// TIA Portal project "PAD_Printer" (V16)

(* hardware
DEVICE "S7-1200 station_1"  S7-1200 Station
   slot 0: "Rack_0"  S7-1200 Rack  Rack  V1.0
   slot 1: "PLC_1"  CPU 1214C DC/DC/DC  6ES7 214-1AG40-0XB0  V4.4
DEVICE "HMI_1"  TP700 Comfort
   slot 0: "HMI_1"  TP700 Comfort  6AV2 124-0GC01-0AX0  16.0.0.0
   slot 1: "HMI_RT_1"  TP700 Comfort  6AV2 124-0GC01-0AX0  16.0.0.0
   slot 5: "HMI_1.IE_CP_1"  PROFINET Interface  16.0.0.0
      slot 1: "PROFINET Interface_1"  PROFINET Interface
         slot 1: "Port_1"  Port
         slot 2: "Port_2"  Port
   slot 7: "HMI_1.MPI/DP_CP_1"  MPI/DP Interface  16.0.0.0
*)

// ===== PLC "PLC_1"  CPU 1214C DC/DC/DC =====

VAR_GLOBAL   // PLC tag table "Default tag table"
   "AUTO" AT %I0.0 : Bool;   // Chế độ Auto
   "MAN" AT %I0.1 : Bool;   // Chế độ Manual
   "FOOT SWITCH" AT %I0.2 : Bool;   // Bàn đạp của chế độ Manual
   "X-CYLINDER IN" AT %I0.3 : Bool;   // Cảm biến xylanh thu về
   "X-CYLINDER OUT" AT %I0.4 : Bool;   // Cảm biến xylanh đi ra
   "Y-CYLINDER UPPER" AT %I0.5 : Bool;   // Cảm biến xylanh bên trên
   "Y-CYLINDER LOWER" AT %I0.6 : Bool;   // Cảm biến xylanh bên dưới
   "CLEAN" AT %I0.7 : Bool;   // Chế độ Clean
   "X-CYLINDER RUN" AT %Q0.0 : Bool;   // Xylanh trục X chạy
   "Y-CYLINDER RUN" AT %Q0.1 : Bool;   // Xylanh trục Y chạy
   "Tag_1" AT %M5.0 : Bool;   // Bit trung gian của chế độ Manual, Auto
   "Tag_2" AT %M5.1 : Bool;   // Bit trung gian của chế độ Manual, Auto
   "Time_delay" AT %M5.2 : Bool;   // Bit trung gian timer của chế độ Auto
   "Tag_3" AT %M5.3 : Bool;   // Bit trung gian của chế độ Manual
   "Tag_4" AT %M5.4 : Bool;   // Bit trung gian của chế độ Auto
   "Tag_5" AT %M5.5 : Bool;   // Bit trung gian của chế độ Auto
   "Tag_6" AT %M5.6 : Bool;   // Bit trung gian của chế độ Auto
   "PV-T" AT %MD100 : DInt;   // Hiển thị thời gian delay trong Auto
   "Tag_7" AT %M6.0 : Bool;   // Bit nhớ của lệnh xung sườn xuống
   "Tag_8" AT %M6.1 : Bool;   // Bit nhớ của lệnh xung sườn xuống
END_VAR

DATA_BLOCK "DATA"   // DB1
{ S7_Optimized_Access := 'FALSE' }
VERSION : 0.1
   VAR
      AUTO : Bool;   // Chế độ Auto
      MAN : Bool;   // Chế độ Manual
      "FOOT SWITCH" : Bool;   // Bàn đạp của chế độ Manual
      "X-CYLINDER IN" : Bool;   // Cảm biến xylanh thu về
      "X-CYLINDER OUT" : Bool;   // Cảm biến xylanh đi ra
      "Y-CYLINDER UPPER" : Bool;   // Cảm biến xylanh bên trên
      "Y-CYLINDER LOWER" : Bool;   // Cảm biến xylanh bên dưới
      CLEAN : Bool;   // Chế độ Clean
      "X-CYLINDER RUN" : Bool;   // Xylanh trục X chạy
      "Y-CYLINDER RUN" : Bool;   // Xylanh trục Y chạy
      Define_Man : Bool;
      Define_Auto : Bool;
      AUTO_I : Bool;
      MAN_I : Bool;
      "FOOT SWITCH_I" : Bool;
      "X-CYLINDER IN_I" : Bool;
      "X_CYLINDER OUT_I" : Bool;
      "Y-CYLINDER UPPER_I" : Bool;
      "Y-CYLINDER LOWER_I" : Bool;
      CLEAN_I : Bool;
      "X-CYLINDER RUN_I" : Bool;
      "Y-CYLINDER RUN_I" : Bool;
      RESETALL : Bool;
   END_VAR
BEGIN
END_DATA_BLOCK

// folder: System blocks/Program resources

DATA_BLOCK "T"   // DB2
{ S7_Optimized_Access := 'TRUE' }
AUTHOR : Simatic
FAMILY : IEC
NAME : IEC_TMR
VERSION : 1.0
// stored: InstanceOfName IEC_TIMER
"IEC_TIMER"
BEGIN
END_DATA_BLOCK

// folder: (top level)

FUNCTION "INPUT" : Void   // FC1, LAD
{ S7_Optimized_Access := 'TRUE' }
VERSION : 0.1
BEGIN

REGION Network 1: Chế độ AUTO
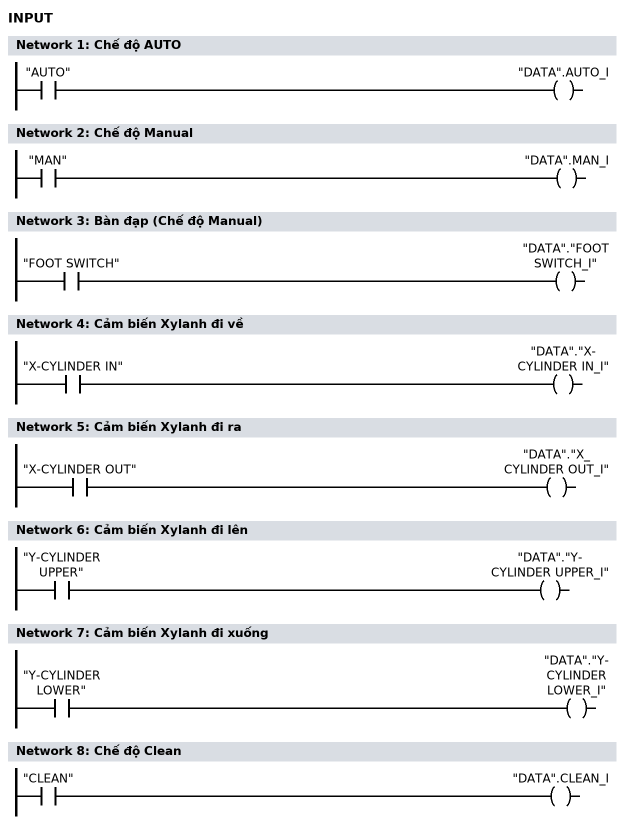
   RUNG wire#powerrail
      Contact( "AUTO" )
      Coil( "DATA".AUTO_I )
   END_RUNG
   // the same network as SCL:
   "DATA".AUTO_I := "AUTO";
END_REGION

REGION Network 2: Chế độ Manual
   RUNG wire#powerrail
      Contact( "MAN" )
      Coil( "DATA".MAN_I )
   END_RUNG
   // the same network as SCL:
   "DATA".MAN_I := "MAN";
END_REGION

REGION Network 3: Bàn đạp (Chế độ Manual)
   RUNG wire#powerrail
      Contact( "FOOT SWITCH" )
      Coil( "DATA"."FOOT SWITCH_I" )
   END_RUNG
   // the same network as SCL:
   "DATA"."FOOT SWITCH_I" := "FOOT SWITCH";
END_REGION

REGION Network 4: Cảm biến Xylanh đi về
   RUNG wire#powerrail
      Contact( "X-CYLINDER IN" )
      Coil( "DATA"."X-CYLINDER IN_I" )
   END_RUNG
   // the same network as SCL:
   "DATA"."X-CYLINDER IN_I" := "X-CYLINDER IN";
END_REGION

REGION Network 5: Cảm biến Xylanh đi ra
   RUNG wire#powerrail
      Contact( "X-CYLINDER OUT" )
      Coil( "DATA"."X_CYLINDER OUT_I" )
   END_RUNG
   // the same network as SCL:
   "DATA"."X_CYLINDER OUT_I" := "X-CYLINDER OUT";
END_REGION

REGION Network 6: Cảm biến Xylanh đi lên
   RUNG wire#powerrail
      Contact( "Y-CYLINDER UPPER" )
      Coil( "DATA"."Y-CYLINDER UPPER_I" )
   END_RUNG
   // the same network as SCL:
   "DATA"."Y-CYLINDER UPPER_I" := "Y-CYLINDER UPPER";
END_REGION

REGION Network 7: Cảm biến Xylanh đi xuống
   RUNG wire#powerrail
      Contact( "Y-CYLINDER LOWER" )
      Coil( "DATA"."Y-CYLINDER LOWER_I" )
   END_RUNG
   // the same network as SCL:
   "DATA"."Y-CYLINDER LOWER_I" := "Y-CYLINDER LOWER";
END_REGION

REGION Network 8: Chế độ Clean
   RUNG wire#powerrail
      Contact( "CLEAN" )
      Coil( "DATA".CLEAN_I )
   END_RUNG
   // the same network as SCL:
   "DATA".CLEAN_I := "CLEAN";
END_REGION
END_FUNCTION

FUNCTION "OUTPUT" : Void   // FC2, LAD
{ S7_Optimized_Access := 'TRUE' }
VERSION : 0.1
BEGIN

REGION Network 1: Chạy Xylanh trục X
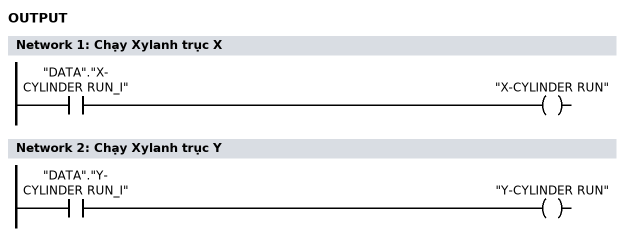
   RUNG wire#powerrail
      Contact( "DATA"."X-CYLINDER RUN_I" )
      Coil( "X-CYLINDER RUN" )
   END_RUNG
   // the same network as SCL:
   "X-CYLINDER RUN" := "DATA"."X-CYLINDER RUN_I";
END_REGION

REGION Network 2: Chạy Xylanh trục Y
   RUNG wire#powerrail
      Contact( "DATA"."Y-CYLINDER RUN_I" )
      Coil( "Y-CYLINDER RUN" )
   END_RUNG
   // the same network as SCL:
   "Y-CYLINDER RUN" := "DATA"."Y-CYLINDER RUN_I";
END_REGION
END_FUNCTION

FUNCTION "Auto_Mode" : Void   // FC3, LAD
{ S7_Optimized_Access := 'TRUE' }
VERSION : 0.1
   VAR_TEMP   // added for the SCL form of the ladder/FBD networks
      _w1 : Bool;
   END_VAR
BEGIN

REGION Network 1: Xác nhận chế độ Auto
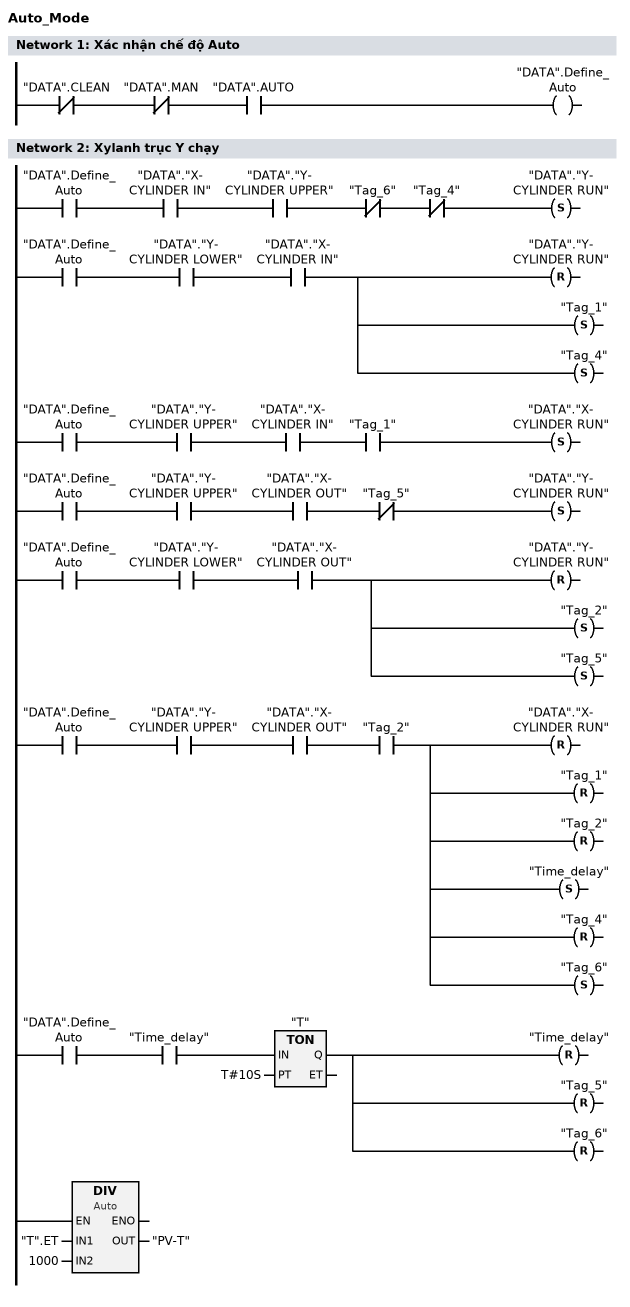
   RUNG wire#powerrail
      I_Contact( "DATA".CLEAN )
      I_Contact( "DATA".MAN )
      Contact( "DATA".AUTO )
      Coil( "DATA".Define_Auto )
   END_RUNG
   // the same network as SCL:
   "DATA".Define_Auto := NOT "DATA".CLEAN AND NOT "DATA".MAN AND "DATA".AUTO;
END_REGION

REGION Network 2: Xylanh trục Y chạy
   IF "DATA".Define_Auto AND "DATA"."X-CYLINDER IN" AND "DATA"."Y-CYLINDER UPPER" AND NOT "Tag_6" AND NOT "Tag_4" THEN
       "DATA"."Y-CYLINDER RUN" := TRUE;
   END_IF;
   IF "DATA".Define_Auto AND "DATA"."Y-CYLINDER LOWER" AND "DATA"."X-CYLINDER IN" THEN
       "DATA"."Y-CYLINDER RUN" := FALSE;
       "Tag_1" := TRUE;
       "Tag_4" := TRUE;
   END_IF;
   IF "DATA".Define_Auto AND "DATA"."Y-CYLINDER UPPER" AND "DATA"."X-CYLINDER IN" AND "Tag_1" THEN
       "DATA"."X-CYLINDER RUN" := TRUE;
   END_IF;
   IF "DATA".Define_Auto AND "DATA"."Y-CYLINDER UPPER" AND "DATA"."X-CYLINDER OUT" AND NOT "Tag_5" THEN
       "DATA"."Y-CYLINDER RUN" := TRUE;
   END_IF;
   IF "DATA".Define_Auto AND "DATA"."Y-CYLINDER LOWER" AND "DATA"."X-CYLINDER OUT" THEN
       "DATA"."Y-CYLINDER RUN" := FALSE;
       "Tag_2" := TRUE;
       "Tag_5" := TRUE;
   END_IF;
   IF "DATA".Define_Auto AND "DATA"."Y-CYLINDER UPPER" AND "DATA"."X-CYLINDER OUT" AND "Tag_2" THEN
       "DATA"."X-CYLINDER RUN" := FALSE;
       "Tag_1" := FALSE;
   END_IF;
   #_w1 := "DATA".Define_Auto AND "DATA"."Y-CYLINDER UPPER" AND "DATA"."X-CYLINDER OUT" AND "Tag_2";
   IF #_w1 THEN
       "Tag_2" := FALSE;
       "Time_delay" := TRUE;
       "Tag_4" := FALSE;
       "Tag_6" := TRUE;
   END_IF;
   "T".TON(IN := "DATA".Define_Auto AND "Time_delay", PT := T#10S);
   IF "T".Q THEN
       "Time_delay" := FALSE;
       "Tag_5" := FALSE;
       "Tag_6" := FALSE;
   END_IF;
   "PV-T" := "T".ET / 1000;
END_REGION
END_FUNCTION

FUNCTION "Man_Mode" : Void   // FC4, LAD
{ S7_Optimized_Access := 'TRUE' }
VERSION : 0.1
BEGIN

REGION Network 1: Xác nhận chế độ Man
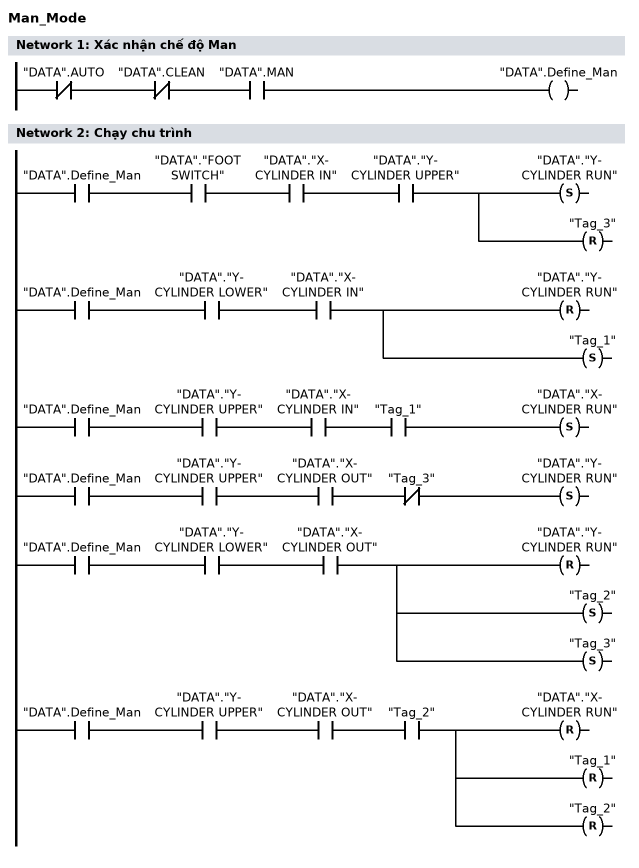
   RUNG wire#powerrail
      I_Contact( "DATA".AUTO )
      I_Contact( "DATA".CLEAN )
      Contact( "DATA".MAN )
      Coil( "DATA".Define_Man )
   END_RUNG
   // the same network as SCL:
   "DATA".Define_Man := NOT "DATA".AUTO AND NOT "DATA".CLEAN AND "DATA".MAN;
END_REGION

REGION Network 2: Chạy chu trình
   RUNG wire#powerrail
      Contact( "DATA".Define_Man )
      Contact( "DATA"."FOOT SWITCH" )
      Contact( "DATA"."X-CYLINDER IN" )
      Contact( "DATA"."Y-CYLINDER UPPER" )
      wire#w1
      S_Coil( "DATA"."Y-CYLINDER RUN" )
   END_RUNG
   RUNG wire#w1
      R_Coil( "Tag_3" )
   END_RUNG
   RUNG wire#powerrail
      Contact( "DATA".Define_Man )
      Contact( "DATA"."Y-CYLINDER LOWER" )
      Contact( "DATA"."X-CYLINDER IN" )
      wire#w2
      R_Coil( "DATA"."Y-CYLINDER RUN" )
   END_RUNG
   RUNG wire#w2
      S_Coil( "Tag_1" )
   END_RUNG
   RUNG wire#powerrail
      Contact( "DATA".Define_Man )
      Contact( "DATA"."Y-CYLINDER UPPER" )
      Contact( "DATA"."X-CYLINDER IN" )
      Contact( "Tag_1" )
      S_Coil( "DATA"."X-CYLINDER RUN" )
   END_RUNG
   RUNG wire#powerrail
      Contact( "DATA".Define_Man )
      Contact( "DATA"."Y-CYLINDER UPPER" )
      Contact( "DATA"."X-CYLINDER OUT" )
      I_Contact( "Tag_3" )
      S_Coil( "DATA"."Y-CYLINDER RUN" )
   END_RUNG
   RUNG wire#powerrail
      Contact( "DATA".Define_Man )
      Contact( "DATA"."Y-CYLINDER LOWER" )
      Contact( "DATA"."X-CYLINDER OUT" )
      wire#w3
      R_Coil( "DATA"."Y-CYLINDER RUN" )
   END_RUNG
   RUNG wire#w3
      S_Coil( "Tag_2" )
   END_RUNG
   RUNG wire#w3
      S_Coil( "Tag_3" )
   END_RUNG
   RUNG wire#powerrail
      Contact( "DATA".Define_Man )
      Contact( "DATA"."Y-CYLINDER UPPER" )
      Contact( "DATA"."X-CYLINDER OUT" )
      Contact( "Tag_2" )
      wire#w4
      R_Coil( "DATA"."X-CYLINDER RUN" )
   END_RUNG
   RUNG wire#w4
      R_Coil( "Tag_1" )
   END_RUNG
   RUNG wire#w4
      R_Coil( "Tag_2" )
   END_RUNG
   // the same network as SCL:
   IF "DATA".Define_Man AND "DATA"."FOOT SWITCH" AND "DATA"."X-CYLINDER IN" AND "DATA"."Y-CYLINDER UPPER" THEN
       "DATA"."Y-CYLINDER RUN" := TRUE;
       "Tag_3" := FALSE;
   END_IF;
   IF "DATA".Define_Man AND "DATA"."Y-CYLINDER LOWER" AND "DATA"."X-CYLINDER IN" THEN
       "DATA"."Y-CYLINDER RUN" := FALSE;
       "Tag_1" := TRUE;
   END_IF;
   IF "DATA".Define_Man AND "DATA"."Y-CYLINDER UPPER" AND "DATA"."X-CYLINDER IN" AND "Tag_1" THEN
       "DATA"."X-CYLINDER RUN" := TRUE;
   END_IF;
   IF "DATA".Define_Man AND "DATA"."Y-CYLINDER UPPER" AND "DATA"."X-CYLINDER OUT" AND NOT "Tag_3" THEN
       "DATA"."Y-CYLINDER RUN" := TRUE;
   END_IF;
   IF "DATA".Define_Man AND "DATA"."Y-CYLINDER LOWER" AND "DATA"."X-CYLINDER OUT" THEN
       "DATA"."Y-CYLINDER RUN" := FALSE;
       "Tag_2" := TRUE;
       "Tag_3" := TRUE;
   END_IF;
   IF "DATA".Define_Man AND "DATA"."Y-CYLINDER UPPER" AND "DATA"."X-CYLINDER OUT" AND "Tag_2" THEN
       "DATA"."X-CYLINDER RUN" := FALSE;
       "Tag_1" := FALSE;
       "Tag_2" := FALSE;
   END_IF;
END_REGION
END_FUNCTION

FUNCTION "Clean_Mode" : Void   // FC5, LAD
{ S7_Optimized_Access := 'TRUE' }
VERSION : 0.1
BEGIN

REGION Network 1: Chế độ Clean
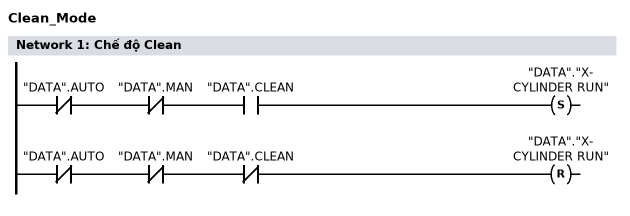
   RUNG wire#powerrail
      I_Contact( "DATA".AUTO )
      I_Contact( "DATA".MAN )
      Contact( "DATA".CLEAN )
      S_Coil( "DATA"."X-CYLINDER RUN" )
   END_RUNG
   RUNG wire#powerrail
      I_Contact( "DATA".AUTO )
      I_Contact( "DATA".MAN )
      I_Contact( "DATA".CLEAN )
      R_Coil( "DATA"."X-CYLINDER RUN" )
   END_RUNG
   // the same network as SCL:
   IF NOT "DATA".AUTO AND NOT "DATA".MAN AND "DATA".CLEAN THEN "DATA"."X-CYLINDER RUN" := TRUE; END_IF;
   IF NOT "DATA".AUTO AND NOT "DATA".MAN AND NOT "DATA".CLEAN THEN "DATA"."X-CYLINDER RUN" := FALSE; END_IF;
END_REGION
END_FUNCTION

ORGANIZATION_BLOCK "Main"   // OB1, LAD, ProgramCycle
TITLE = "Main Program Sweep (Cycle)"
{ S7_Optimized_Access := 'TRUE' }
VERSION : 0.1
   VAR_INPUT
      Initial_Call : Bool;   // Initial call of this OB
      Remanence : Bool;   // =True, if remanent data are available
   END_VAR
   VAR_TEMP   // added for the SCL form of the ladder/FBD networks
      _w1 : Bool;
      _w2 : Bool;
   END_VAR
BEGIN

REGION Network 1: Input
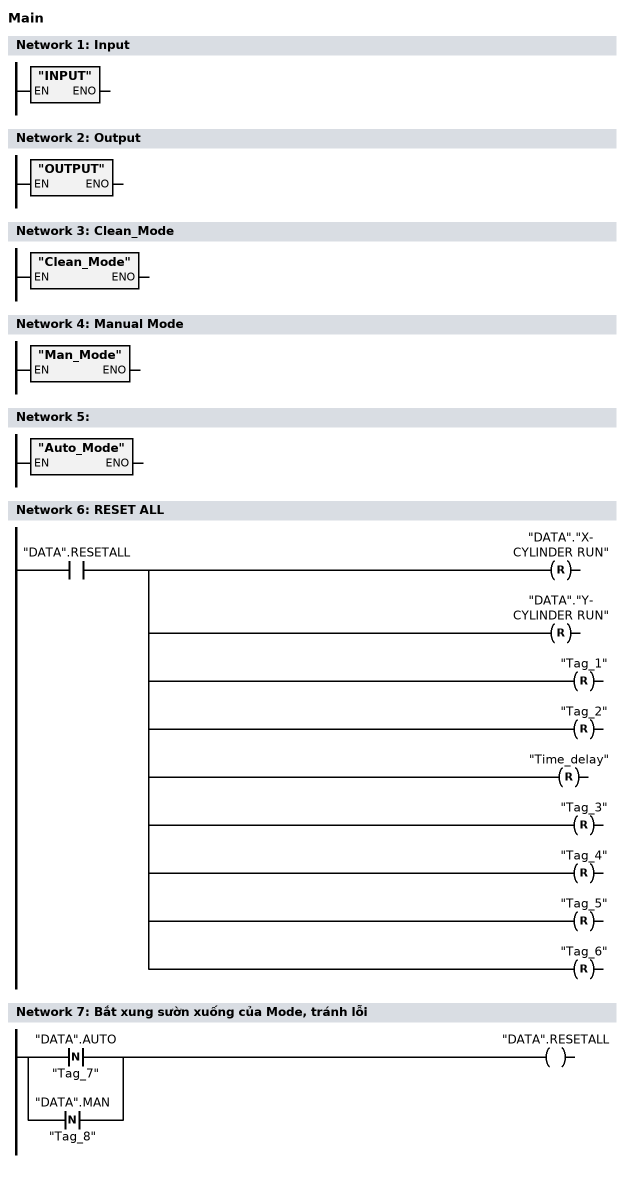
   RUNG wire#powerrail
      "INPUT"()
   END_RUNG
   // the same network as SCL:
   "INPUT"();
END_REGION

REGION Network 2: Output
   RUNG wire#powerrail
      "OUTPUT"()
   END_RUNG
   // the same network as SCL:
   "OUTPUT"();
END_REGION

REGION Network 3: Clean_Mode
   RUNG wire#powerrail
      "Clean_Mode"()
   END_RUNG
   // the same network as SCL:
   "Clean_Mode"();
END_REGION

REGION Network 4: Manual Mode
   RUNG wire#powerrail
      "Man_Mode"()
   END_RUNG
   // the same network as SCL:
   "Man_Mode"();
END_REGION

REGION Network 5
   RUNG wire#powerrail
      "Auto_Mode"()
   END_RUNG
   // the same network as SCL:
   "Auto_Mode"();
END_REGION

REGION Network 6: RESET ALL
   RUNG wire#powerrail
      Contact( "DATA".RESETALL )
      wire#w1
      R_Coil( "DATA"."X-CYLINDER RUN" )
   END_RUNG
   RUNG wire#w1
      R_Coil( "DATA"."Y-CYLINDER RUN" )
   END_RUNG
   RUNG wire#w1
      R_Coil( "Tag_1" )
   END_RUNG
   RUNG wire#w1
      R_Coil( "Tag_2" )
   END_RUNG
   RUNG wire#w1
      R_Coil( "Time_delay" )
   END_RUNG
   RUNG wire#w1
      R_Coil( "Tag_3" )
   END_RUNG
   RUNG wire#w1
      R_Coil( "Tag_4" )
   END_RUNG
   RUNG wire#w1
      R_Coil( "Tag_5" )
   END_RUNG
   RUNG wire#w1
      R_Coil( "Tag_6" )
   END_RUNG
   // the same network as SCL:
   IF "DATA".RESETALL THEN
       "DATA"."X-CYLINDER RUN" := FALSE;
       "DATA"."Y-CYLINDER RUN" := FALSE;
       "Tag_1" := FALSE;
       "Tag_2" := FALSE;
       "Time_delay" := FALSE;
       "Tag_3" := FALSE;
       "Tag_4" := FALSE;
       "Tag_5" := FALSE;
       "Tag_6" := FALSE;
   END_IF;
END_REGION

REGION Network 7: Bắt xung sườn xuống của Mode, tránh lỗi
   RUNG wire#powerrail
      N_Contact(operand := "DATA".AUTO, bit := "Tag_7")
      wire#w1
      Coil( "DATA".RESETALL )
   END_RUNG
   RUNG wire#powerrail
      N_Contact(operand := "DATA".MAN, bit := "Tag_8")
   END_RUNG wire#w1
   // the same network as SCL:
   #_w1 := NOT "DATA".AUTO AND "Tag_7";   // falling edge of "DATA".AUTO
   "Tag_7" := "DATA".AUTO;
   #_w2 := NOT "DATA".MAN AND "Tag_8";   // falling edge of "DATA".MAN
   "Tag_8" := "DATA".MAN;
   "DATA".RESETALL := #_w1 OR #_w2;
END_REGION
END_ORGANIZATION_BLOCK

(* ===== HMI "HMI_RT_1" =====
system functions are stored by id; their names below are inferred from use
connection "HMI_Connection_1": ETHERNET, S7_1200_OMS
connection "HMI_Connection_2": ETHERNET, S7_1200_OMS

HMI tags "Default tag table"
   "DATA_AUTO" : Bool = PLC DATA.AUTO AT %DB1.DBX0.0, 1 s
   "DATA_MAN" : Bool = PLC DATA.MAN AT %DB1.DBX0.1, 1 s
   "DATA_CLEAN" : Bool = PLC DATA.CLEAN AT %DB1.DBX0.7, 1 s
   "DATA_RESETALL" : Bool = PLC DATA.RESETALL AT %DB1.DBX2.6, 1 s
   "DATA_FOOT SWITCH" : Bool = PLC DATA."FOOT SWITCH" AT %DB1.DBX0.2, 1 s
   "DATA_Y-CYLINDER UPPER" : Bool = PLC DATA."Y-CYLINDER UPPER" AT %DB1.DBX0.5, 1 s
   "DATA_Y-CYLINDER LOWER" : Bool = PLC DATA."Y-CYLINDER LOWER" AT %DB1.DBX0.6, 1 s
   "DATA_X-CYLINDER IN" : Bool = PLC DATA."X-CYLINDER IN" AT %DB1.DBX0.3, 1 s
   "DATA_X-CYLINDER OUT" : Bool = PLC DATA."X-CYLINDER OUT" AT %DB1.DBX0.4, 1 s
   "DATA_Y-CYLINDER RUN" : Bool = PLC DATA."Y-CYLINDER RUN" AT %DB1.DBX1.1, 1 s
   "DATA_X-CYLINDER RUN" : Bool = PLC DATA."X-CYLINDER RUN" AT %DB1.DBX1.0, 1 s
   "PV-T" : DInt = PLC "PV-T" AT %MD100, 1 s

screen "Root screen" 800x480, template "Template_1"
   TextField "HmiScreenItemData" at 80,196 size 640x25; Text 'Welcome to HMI_1 (TP700 Comfort)!'

Template "Template_1" 800x480
   Button "Exit" at 720,420 size 78x58; TextOff 'Exit'; PictureOff "ExitRuntime_TP700_Comfort_TR"; PictureOn "ExitRuntime_TP700_Comfort_TR"
      on Release: StopRuntime(0)
   Button "Template_Button" at 640,420 size 78x58; TextOff 'Text'
   Button "Template_Button_1" at 560,420 size 78x58; TextOff 'Text'
   Button "Template_Button_2" at 480,420 size 78x58; TextOff 'Text'
   Button "Template_Button_3" at 400,420 size 78x58; TextOff 'Text'
   Button "Template_Button_4" at 321,420 size 78x58; TextOff 'Text'
   Button "Template_Button_5" at 241,420 size 78x58; TextOff 'Text'
   Button "Template_Button_6" at 161,420 size 78x58; TextOff 'Text'
   Button "Template_Button_7" at 81,420 size 78x58; TextOff 'Text'
   Button "Start screen" at 1,420 size 78x58; TextOff 'Start screen'; PictureOff "NavigateHome_TP700_Comfort_TR"; PictureOn "NavigateHome_TP700_Comfort_TR"
      on Release: ActivateScreen("Root screen", 0)

screen "Screen_1" 800x480
   Button "Button_1" at 25,16 size 96x32; TextOff 'AUTO'
      on Click: InvertBit("DATA_AUTO")
      Appearance <- "DATA_AUTO"
   SymbolLibrary "Symbol library_1" at 35,249 size 256x24
      Visibility <- "DATA_X-CYLINDER RUN"
   SymbolLibrary "Symbol library_2" at 34,250 size 457x25
      Visibility <- "DATA_X-CYLINDER RUN"
   SymbolLibrary "Symbol library_3" at 200,210 size 67x19
      on Click: InvertBit("DATA_Y-CYLINDER UPPER")
      Appearance <- "DATA_Y-CYLINDER UPPER"
   IOField "I/O field_1" at 677,150 size 96x32; FormatPattern 1
      ProcessValue <- "DATA_X-CYLINDER RUN"
   TextField "Text field_1" at 590,159 size 84x23; Text 'Xylanh X'
   Button "Button_3" at 161,16 size 96x32; TextOff 'MAN'
      on Click: InvertBit("DATA_MAN")
      Appearance <- "DATA_MAN"
   Button "Button_4" at 300,16 size 96x32; TextOff 'CLEAN'
      on Click: InvertBit("DATA_CLEAN")
      Appearance <- "DATA_CLEAN"
   Button "Button_5" at 433,16 size 123x32; TextOff 'FOOTSWITCH'
      on Release: ResetBit("DATA_FOOT SWITCH")
      on Press: SetBit("DATA_FOOT SWITCH")
      Appearance <- "DATA_FOOT SWITCH"
   SymbolLibrary "Symbol library_4" at 195,342 size 67x19
      on Click: InvertBit("DATA_Y-CYLINDER LOWER")
      Appearance <- "DATA_Y-CYLINDER LOWER"
   SymbolLibrary "Symbol library_5" at 271,135 size 19x67
      on Click: InvertBit("DATA_X-CYLINDER IN")
      Appearance <- "DATA_X-CYLINDER IN"
   SymbolLibrary "Symbol library_6" at 473,134 size 19x67
      on Click: InvertBit("DATA_X-CYLINDER OUT")
      Appearance <- "DATA_X-CYLINDER OUT"
   SymbolLibrary "Symbol library_7" at 300,60 size 24x169
      Visibility <- "DATA_Y-CYLINDER RUN"
   SymbolLibrary "Symbol library_8" at 299,58 size 25x305
      Visibility <- "DATA_Y-CYLINDER RUN"
   TextField "Text field_2" at 286,418 size 69x23; Text 'Lọ mực'
   TextField "Text field_3" at 451,418 size 93x23; Text 'Sản phẩm'
   TextField "Text field_4" at 589,211 size 84x23; Text 'Xylanh Y'
   IOField "I/O field_2" at 679,201 size 96x32; FormatPattern 1
      ProcessValue <- "DATA_Y-CYLINDER RUN"
   IOField "I/O field_3" at 685,275 size 96x32; FormatPattern 999
      ProcessValue <- "PV-T"
*)